(* CoDeSys 2.3.9.41 project: plcprob1.pro *)
(* Libraries: Standard.lib 4.10.05 11:14:46, IecSfc.lib 13.4.06 15:51:28, SYSLIBCALLBACK.LIB 26.9.08 16:43:52 *)

(* POU PLC_PRG, ST *)
PROGRAM PLC_PRG
VAR
	Counter: INT;
	X_pos: INT;
	ext:BOOL;
	myTON:TON;
END_VAR
X_pos:=0;
ext:=TRUE;
WHILE X_pos<100 DO
	X_pos:=X_pos+1;
	myTON(IN:=ext , PT:= t#1s);
END_WHILE;
RETURN;
END_PROGRAM

(* Visualisation observer
rectangle at (120,130)-(191,181): x offset PLC_PRG.X_pos
*)
